TYPE ST_LaudaWriteCommands_Rights :
STRUCT
	KeyboardMaster_UlockLock				: STRING := 'OUT_MODE_00_';
	KeyboardRemoveControlUnit_UnlockLock	: STRING := 'OUT_MODE_03_X';
	
END_STRUCT
END_TYPE

(* stored: Version 1.1.0.1, ProductVersion 3.1.4024.12
   DUT ST_LaudaWriteCommands_Rights: Id {9469727b-78cc-436d-9be4-f146139396d1} *)
